FUNCTION_BLOCK AxisAbsTestSuite
VAR
	StubAxis : AXIS_REF;
	iStubTask : I_Task;
	TestAxisAbs : MoveAbsTask := (AxisRef := stubaxis);
	TestObjRunner : ObjectRunner<99>;
	ObjTestSuite : TestSuite<TestSuiteParameter.MaxTestCount>('C:\ProgramData\Beckhoff\TwinCAT\3.1\Boot\Object_Tests.xml') := (TestSuiteName := 'Object Test Suite');
END_VAR

CheckCorrectRegistration_Test();
TaskAcceptValidCommand_Test();
TaskRejectsZeroVeloCommand_Test();

METHOD CheckCorrectRegistration_Test : BOOL
VAR_INST
	Expected : BOOL := TRUE;
	Actual	 : bool;
END_VAR
IF ObjTestSuite.Test(__POUNAME()).ExecuteTest() THEN
	TestAxisAbs.RegisterWithParent(TestObjRunner);
	Actual := TestObjRunner.CyclicModuleCount = TestObjRunner.AbortableModuleCount AND
				TestObjRunner.CyclicModuleCount = TestObjRunner.TaskModuleCount;
	ObjTestSuite.Test(__POUNAME()).AssertEqual(Expected, Actual);
END_IF
END_METHOD

METHOD TaskAcceptValidCommand_Test : BOOL
VAR_INST
	Expected : BOOL := TRUE;
	Actual	 : BOOL;
END_VAR
IF ObjTestSuite.Test(__POUNAME()).ExecuteTest() THEN
	Actual := SUCCEEDED(TestAxisAbs.MoveTo(100.0, 300.0));
	TestAxisAbs.Abort();
	ObjTestSuite.Test(__POUNAME()).AssertEqual(Expected, Actual);
END_IF
END_METHOD

METHOD TaskRejectsZeroVeloCommand_Test : BOOL
VAR_INST
	Expected : BOOL := TRUE;
	Actual	 : BOOL;
END_VAR
IF ObjTestSuite.Test(__POUNAME()).ExecuteTest() THEN
	Actual := FAILED(TestAxisAbs.MoveTo(100.0, 0.0));
	TestAxisAbs.Abort();
	ObjTestSuite.Test(__POUNAME()).AssertEqual(Expected, Actual);
END_IF
END_METHOD

END_FUNCTION_BLOCK

(* stored: Version 1.1.0.1
   POU AxisAbsTestSuite: Id {931c3bf4-e690-4ab0-bb8d-cbf096b9e190}, SpecialFunc None
   Method CheckCorrectRegistration_Test: Id {c4385ca2-d3df-42c8-9370-a356405e0465}
   Method TaskAcceptValidCommand_Test: Id {d5bc1b43-cf1a-4b0e-b9f0-4a82dce35f41}
   Method TaskRejectsZeroVeloCommand_Test: Id {6092ced4-346a-4b46-85f8-d8b449d061cc} *)
